(* CODESYS project Motor_Control_TM241CE40T.project
   Author: PLCAutoPilot
   Version: 0.0.0.0
   Description: Motor Start/Stop with Overload Alarm
   Title: Motor_Control_Station
   Company: PLCAutoPilot

Project tree, tasks and I/O mapping:
  M241_Motor_Control : TM241CE40T/U, Schneider Electric, order no. TM241CE40T/U, version 5.0.8.2
    Application
      task TASK_SR_MainMachine (cyclic, interval t#10ms, priority 8, watchdog t#10ms x 10) calls SR_MainMachine
      task TASK_SR_Diagnostics (cyclic, interval t#100ms, priority 31, watchdog t#100ms x 10) calls SR_Diagnostics
      Module Manager
    DI : Digital Inputs, Schneider Electric, version 5.0.8.2
        input  idwDI_IDW0 : DWORD  // IDW0
        input  ibDI_IB1 : BYTE  // IB1
    DQ : Digital Outputs, Schneider Electric, version 5.0.8.2
        output qwDQ_QW0 : WORD  // QW0
        output qbDQ_QB1 : BYTE  // QB1
    Counters : Counters, Schneider Electric, version 5.0.8.2
    Pulse_Generators : Pulse Generators, Schneider Electric, version 5.0.8.2
    Cartridge_1 : Cartridge, Schneider Electric, version 5.0.8.2
    Cartridge_2 : Cartridge, Schneider Electric, version 5.0.8.2
    IO_Bus : IO bus - TM3, Schneider Electric, version 5.0.8.2
    COM_Bus : COM bus, Schneider Electric, version 5.0.8.2
    Ethernet_1 : Ethernet Network, Schneider Electric, version 5.0.8.2
    Serial_Line_1 : Serial line, Schneider Electric, version 5.0.8.2
      Machine_Expert_Network_Manager : Machine Expert-Network Manager, Schneider Electric, version 4.0.0.3
    Serial_Line_2 : Serial line, Schneider Electric, version 5.0.8.2
      Modbus_Manager : Modbus Manager, Schneider Electric, version 4.0.0.3
  MainMachine
    Module Interface
    CommandList
    OperationModeManagement
      Auto
    TemplateExceptions
    TemplateReactions
    text StopEndOfCycle
    text StopNow
    Infrastructure
      TemplateGlobalReactions
  MainMachine
  program PLC_PRG [LD]
*)

// PLC_PRG
PROGRAM PLC_PRG
VAR
	///Emergency Stop Push Button (NC - Normally Closed)
	EMERGENCY_PB AT %IX0.0: BOOL;
	///Start Push Button (NO - Normally Open)
	START_PB AT %IX0.1: BOOL;
	///Stop Push Button (NC - Normally Closed)
	STOP_PB AT %IX0.2: BOOL;
	///Motor Overload Relay Contact (NC - Normally Closed)
	MOTOR_OL AT %IX0.3: BOOL;
	///Alarm Reset Push Button (NO - Normally Open)
	RESET_PB AT %IX0.4: BOOL;
	///Motor Contactor Output
	MOTOR_RUN AT %QX0.0: BOOL;
	///Motor Running Indicator Lamp
	MOTOR_LAMP AT %QX0.1: BOOL;
	///Overload Alarm Indicator Lamp
	OL_ALARM_LAMP AT %QX0.2: BOOL;
	///System Ready Indicator Lamp
	READY_LAMP AT %QX0.3: BOOL;
	///System Ready Flag - Set after 3 second startup delay
	System_ready AT %M?0: BOOL;
	///Motor Seal-in Memory Bit
	Motor_sealed AT %M?1: BOOL;
	///Overload Alarm Latched Memory Bit
	OL_Alarm_latched AT %M?2: BOOL;
	///3 second startup delay timer
	TON_Startup: TON;
END_VAR

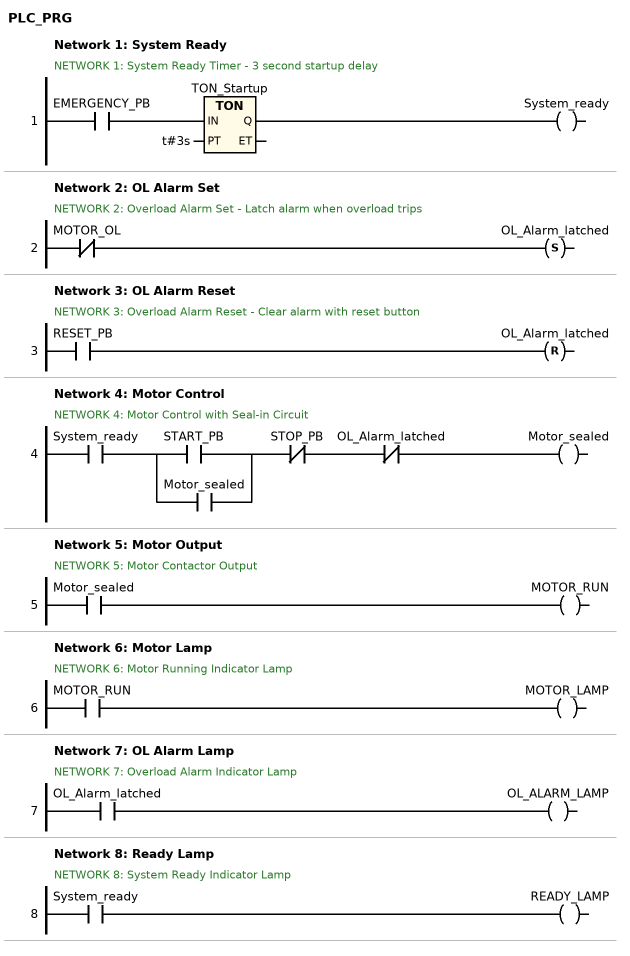
// NETWORK 1: Network 1: System Ready
// NETWORK 1: System Ready Timer - 3 second startup delay
TON_Startup(IN := EMERGENCY_PB, PT := t#3s); // TON
System_ready := TON_Startup.Q;

// NETWORK 2: Network 2: OL Alarm Set
// NETWORK 2: Overload Alarm Set - Latch alarm when overload trips
OL_Alarm_latched S= NOT MOTOR_OL;

// NETWORK 3: Network 3: OL Alarm Reset
// NETWORK 3: Overload Alarm Reset - Clear alarm with reset button
OL_Alarm_latched R= RESET_PB;

// NETWORK 4: Network 4: Motor Control
// NETWORK 4: Motor Control with Seal-in Circuit
Motor_sealed := System_ready AND (START_PB OR Motor_sealed) AND NOT STOP_PB AND NOT OL_Alarm_latched;

// NETWORK 5: Network 5: Motor Output
// NETWORK 5: Motor Contactor Output
MOTOR_RUN := Motor_sealed;

// NETWORK 6: Network 6: Motor Lamp
// NETWORK 6: Motor Running Indicator Lamp
MOTOR_LAMP := MOTOR_RUN;

// NETWORK 7: Network 7: OL Alarm Lamp
// NETWORK 7: Overload Alarm Indicator Lamp
OL_ALARM_LAMP := OL_Alarm_latched;

// NETWORK 8: Network 8: Ready Lamp
// NETWORK 8: System Ready Indicator Lamp
READY_LAMP := System_ready;

END_PROGRAM

(* text StopEndOfCycle
iq_stReactions.xStopEndOfCycle
*)

(* text StopNow
iq_stReactions.xAsyncStop OR iq_stReactions.xSyncStopEl OR iq_stReactions.xSyncStopEh
*)
